FUNCTION_BLOCK Test_TStreamAdd_Read_LREAL EXTENDS TUnitTestBase
VAR
    Stream : TStream(StreamLength := 2);
END_VAR



Stream.Init(2);

Stream.Add_LREAL(1.234567891234);
    
Assertion.AssertEquals_UDINT(
    Expected := 8,
    Actual := Stream.Position,
    VariableName := 'Stream.Position');
    
Stream.Seek(0);

Assertion.AssertEquals_LREAL(
    Expected := 1.234567891234,
    Actual := Stream.Read_LREAL(),
    Delta  := 0.000000000001,
    VariableName := 'Stream.Read_LREAL()');
    
Assertion.AssertEquals_UDINT(
    Expected := 8,
    Actual := Stream.Position,
    VariableName := 'Stream.Position');
    
    
TestFinished();

END_FUNCTION_BLOCK

(* stored: Version 1.1.0.1, ProductVersion 3.1.4024.4
   POU Test_TStreamAdd_Read_LREAL: Id {42a19cb4-2b05-401b-a172-81e8c8a406c3}, SpecialFunc None *)
